{attribute 'GeneratedUsingTerminal: EL6021--0000'}
{attribute addProperty BoxType "EL6021--0000"}
{attribute addProperty Description "EL6021 Interface (RS422/485)"}
{attribute addProperty Physics "KK"}
{attribute addProperty Id "InputsAT %I*Inputs_6C2FC20224OutputsAT %Q*Outputs_5D00B5E724WcStateAT %I*WcState_9091E0EB2InfoDataAT %I*InfoData_32EB74EA10"}
{attribute addProperty CRC "3316510622"}
{attribute addProperty Size "60"}
TYPE EL6021_C5ADEF9E EXTENDS EtcSlaveTerminalBase_947E5A46 :
STRUCT
	{attribute addProperty Name "Inputs"}
	Inputs : Inputs_6C2FC202;
	{attribute addProperty Name "Outputs"}
	Outputs : Outputs_5D00B5E7;
	{attribute addProperty Name "WcState"}
	WcState : WcState_9091E0EB;
	{attribute addProperty Name "InfoData"}
	InfoData : InfoData_32EB74EA;
END_STRUCT
END_TYPE

(* stored: Version 1.2.0.0, ProductVersion 3.1.4024.11
   DUT EL6021_C5ADEF9E: Id {96a66f31-760c-4b2e-ab54-81df9ec3cf45} *)
